// TIA Portal V17 export
// export: Created 2025-03-05T07:59:00.9677921Z, ExportSetting WithDefaults, DisplayName Totally Integrated Automation Portal, DisplayVersion V17 Update 8, DisplayName TIA Portal Openness, DisplayVersion V17 Update 8, DisplayName TIA Portal Version Control Interface, DisplayVersion V17, DisplayName SINAMICS Startdrive Advanced, DisplayVersion V17 SP2, DisplayName SINAMICS Startdrive G110M, G120, G120C, G120D, G120P, G115D, DisplayVersion V17 SP2, DisplayName SINAMICS Startdrive G130, G150, S120, S150, SINAMICS MV, S210, DisplayVersion V17 SP2, DisplayName STEP 7 Professional, DisplayVersion V17 Update 8, DisplayName SINUMERIK ONE STEP 7 Toolbox, DisplayVersion V17 Update 12, DisplayName SINUMERIK 840D sl STEP 7 Toolbox, DisplayVersion V17 Update 12, DisplayName STEP 7 Safety, DisplayVersion V17 Update 6, DisplayName WinCC Advanced, DisplayVersion V17 Update 8
DATA_BLOCK "DB2420_CNC_PLC_SIGNALS"   // DB2420
{ S7_Optimized_Access := 'FALSE'; DB_Accessible_From_OPC_UA := 'FALSE' }
AUTHOR : ETXETAR
VERSION : 1.0
// stored: AutoNumber false, DBAccessibleFromOPCUA false, DBAccessibleFromWebserver true, IsOnlyStoredInLoadMemory false, IsWriteProtectedInAS false
   VAR RETAIN
      NC_PLC_SIGNALS_1_32 : Struct   // NCK INPUTS EXTENSION BIT 41-72 / NC PLC SIGNALS BIT 1-32
         NC_PLC_SIGNAL_1 : Bool;   // NCK INPUTS EXTENSION 41 / UNIT 1 FIXTURE 1 GRIPPER CLOSED
         NC_PLC_SIGNAL_2 : Bool;   // NCK INPUTS EXTENSION 42 / UNIT 1 FIXTURE 1 GRIPPER OPEN
         NC_PLC_SIGNAL_3 : Bool;   // NCK INPUTS EXTENSION 43 / UNIT 1 FIXTURE 1 GRIPPER LOW
         NC_PLC_SIGNAL_4 : Bool;   // NCK INPUTS EXTENSION 44
         NC_PLC_SIGNAL_5 : Bool;   // NCK INPUTS EXTENSION 45
         NC_PLC_SIGNAL_6 : Bool;   // NCK INPUTS EXTENSION 46
         NC_PLC_SIGNAL_7 : Bool;   // NCK INPUTS EXTENSION 47
         NC_PLC_SIGNAL_8 : Bool;   // NCK INPUTS EXTENSION 48
         NC_PLC_SIGNAL_9 : Bool;   // NCK INPUTS EXTENSION 49
         NC_PLC_SIGNAL_10 : Bool;   // NCK INPUTS EXTENSION 50
         NC_PLC_SIGNAL_11 : Bool;   // NCK INPUTS EXTENSION 51
         NC_PLC_SIGNAL_12 : Bool;   // NCK INPUTS EXTENSION 52
         NC_PLC_SIGNAL_13 : Bool;   // NCK INPUTS EXTENSION 53
         NC_PLC_SIGNAL_14 : Bool;   // NCK INPUTS EXTENSION 54
         NC_PLC_SIGNAL_15 : Bool;   // NCK INPUTS EXTENSION 55
         NC_PLC_SIGNAL_16 : Bool;   // NCK INPUTS EXTENSION 56
         NC_PLC_SIGNAL_17 : Bool;   // NCK INPUTS EXTENSION 57 / UNIT 1 FIXTURE 2 GRIPPER CLOSED
         NC_PLC_SIGNAL_18 : Bool;   // NCK INPUTS EXTENSION 58 / UNIT 1 FIXTURE 2 GRIPPER OPEN
         NC_PLC_SIGNAL_19 : Bool;   // NCK INPUTS EXTENSION 59 / UNIT 1 FIXTURE 2 GRIPPER LOW
         NC_PLC_SIGNAL_20 : Bool;   // NCK INPUTS EXTENSION 60
         NC_PLC_SIGNAL_21 : Bool;   // NCK INPUTS EXTENSION 61
         NC_PLC_SIGNAL_22 : Bool;   // NCK INPUTS EXTENSION 62
         NC_PLC_SIGNAL_23 : Bool;   // NCK INPUTS EXTENSION 63
         NC_PLC_SIGNAL_24 : Bool;   // NCK INPUTS EXTENSION 64
         NC_PLC_SIGNAL_25 : Bool;   // NCK INPUTS EXTENSION 65
         NC_PLC_SIGNAL_26 : Bool;   // NCK INPUTS EXTENSION 66
         NC_PLC_SIGNAL_27 : Bool;   // NCK INPUTS EXTENSION 67
         NC_PLC_SIGNAL_28 : Bool;   // NCK INPUTS EXTENSION 68
         NC_PLC_SIGNAL_29 : Bool;   // NCK INPUTS EXTENSION 69
         NC_PLC_SIGNAL_30 : Bool;   // NCK INPUTS EXTENSION 70
         NC_PLC_SIGNAL_31 : Bool;   // NCK INPUTS EXTENSION 71
         NC_PLC_SIGNAL_32 : Bool;   // NCK INPUTS EXTENSION 72
      END_STRUCT;
      NC_PLC_SIGNALS_33_64 : Struct   // NCK INPUTS EXTENSION BIT 73-104 / NC PLC SIGNALS BIT 33-64
         NC_PLC_SIGNAL_33 : Bool;   // NCK INPUTS EXTENSION 73 / UNIT 1 FIXTURE 3 GRIPPER CLOSED
         NC_PLC_SIGNAL_34 : Bool;   // NCK INPUTS EXTENSION 74 / UNIT 1 FIXTURE 3 GRIPPER OPEN
         NC_PLC_SIGNAL_35 : Bool;   // NCK INPUTS EXTENSION 75 / UNIT 1 FIXTURE 3 GRIPPER LOW
         NC_PLC_SIGNAL_36 : Bool;   // NCK INPUTS EXTENSION 76
         NC_PLC_SIGNAL_37 : Bool;   // NCK INPUTS EXTENSION 77
         NC_PLC_SIGNAL_38 : Bool;   // NCK INPUTS EXTENSION 78
         NC_PLC_SIGNAL_39 : Bool;   // NCK INPUTS EXTENSION 79
         NC_PLC_SIGNAL_40 : Bool;   // NCK INPUTS EXTENSION 80
         NC_PLC_SIGNAL_41 : Bool;   // NCK INPUTS EXTENSION 81
         NC_PLC_SIGNAL_42 : Bool;   // NCK INPUTS EXTENSION 82
         NC_PLC_SIGNAL_43 : Bool;   // NCK INPUTS EXTENSION 83
         NC_PLC_SIGNAL_44 : Bool;   // NCK INPUTS EXTENSION 84
         NC_PLC_SIGNAL_45 : Bool;   // NCK INPUTS EXTENSION 85
         NC_PLC_SIGNAL_46 : Bool;   // NCK INPUTS EXTENSION 86
         NC_PLC_SIGNAL_47 : Bool;   // NCK INPUTS EXTENSION 87
         NC_PLC_SIGNAL_48 : Bool;   // NCK INPUTS EXTENSION 88
         NC_PLC_SIGNAL_49 : Bool;   // NCK INPUTS EXTENSION 89 / UNIT 1 FIXTURE 4 GRIPPER CLOSED
         NC_PLC_SIGNAL_50 : Bool;   // NCK INPUTS EXTENSION 90 / UNIT 1 FIXTURE 4 GRIPPER OPEN
         NC_PLC_SIGNAL_51 : Bool;   // NCK INPUTS EXTENSION 91 / UNIT 1 FIXTURE 4 GRIPPER LOW
         NC_PLC_SIGNAL_52 : Bool;   // NCK INPUTS EXTENSION 92
         NC_PLC_SIGNAL_53 : Bool;   // NCK INPUTS EXTENSION 93
         NC_PLC_SIGNAL_54 : Bool;   // NCK INPUTS EXTENSION 94
         NC_PLC_SIGNAL_55 : Bool;   // NCK INPUTS EXTENSION 95
         NC_PLC_SIGNAL_56 : Bool;   // NCK INPUTS EXTENSION 96
         NC_PLC_SIGNAL_57 : Bool;   // NCK INPUTS EXTENSION 97
         NC_PLC_SIGNAL_58 : Bool;   // NCK INPUTS EXTENSION 98
         NC_PLC_SIGNAL_59 : Bool;   // NCK INPUTS EXTENSION 99
         NC_PLC_SIGNAL_60 : Bool;   // NCK INPUTS EXTENSION 100
         NC_PLC_SIGNAL_61 : Bool;   // NCK INPUTS EXTENSION 101
         NC_PLC_SIGNAL_62 : Bool;   // NCK INPUTS EXTENSION 102
         NC_PLC_SIGNAL_63 : Bool;   // NCK INPUTS EXTENSION 103
         NC_PLC_SIGNAL_64 : Bool;   // NCK INPUTS EXTENSION 104
      END_STRUCT;
      NC_PLC_SIGNALS_65_96 : Struct   // NCK INPUTS EXTENSION BIT 73-104 / NC PLC SIGNALS BIT 65-96
         NC_PLC_SIGNAL_65 : Bool;   // NCK INPUTS EXTENSION 73 / UNIT 2 FIXTURE 1 GRIPPER CLOSED
         NC_PLC_SIGNAL_66 : Bool;   // NCK INPUTS EXTENSION 74 / UNIT 2 FIXTURE 1 GRIPPER OPEN
         NC_PLC_SIGNAL_67 : Bool;   // NCK INPUTS EXTENSION 75 / UNIT 2 FIXTURE 1 GRIPPER LOW
         NC_PLC_SIGNAL_68 : Bool;   // NCK INPUTS EXTENSION 76
         NC_PLC_SIGNAL_69 : Bool;   // NCK INPUTS EXTENSION 77
         NC_PLC_SIGNAL_70 : Bool;   // NCK INPUTS EXTENSION 78
         NC_PLC_SIGNAL_71 : Bool;   // NCK INPUTS EXTENSION 79
         NC_PLC_SIGNAL_72 : Bool;   // NCK INPUTS EXTENSION 80
         NC_PLC_SIGNAL_73 : Bool;   // NCK INPUTS EXTENSION 81
         NC_PLC_SIGNAL_74 : Bool;   // NCK INPUTS EXTENSION 82
         NC_PLC_SIGNAL_75 : Bool;   // NCK INPUTS EXTENSION 83
         NC_PLC_SIGNAL_76 : Bool;   // NCK INPUTS EXTENSION 84
         NC_PLC_SIGNAL_77 : Bool;   // NCK INPUTS EXTENSION 85
         NC_PLC_SIGNAL_78 : Bool;   // NCK INPUTS EXTENSION 86
         NC_PLC_SIGNAL_79 : Bool;   // NCK INPUTS EXTENSION 87
         NC_PLC_SIGNAL_80 : Bool;   // NCK INPUTS EXTENSION 88
         NC_PLC_SIGNAL_81 : Bool;   // NCK INPUTS EXTENSION 89 / UNIT 2 FIXTURE 2 GRIPPER CLOSED
         NC_PLC_SIGNAL_82 : Bool;   // NCK INPUTS EXTENSION 90 / UNIT 2 FIXTURE 2 GRIPPER OPEN
         NC_PLC_SIGNAL_83 : Bool;   // NCK INPUTS EXTENSION 91 / UNIT 2 FIXTURE 2 GRIPPER LOW
         NC_PLC_SIGNAL_84 : Bool;   // NCK INPUTS EXTENSION 92
         NC_PLC_SIGNAL_85 : Bool;   // NCK INPUTS EXTENSION 93
         NC_PLC_SIGNAL_86 : Bool;   // NCK INPUTS EXTENSION 94
         NC_PLC_SIGNAL_87 : Bool;   // NCK INPUTS EXTENSION 95
         NC_PLC_SIGNAL_88 : Bool;   // NCK INPUTS EXTENSION 96
         NC_PLC_SIGNAL_89 : Bool;   // NCK INPUTS EXTENSION 97
         NC_PLC_SIGNAL_90 : Bool;   // NCK INPUTS EXTENSION 98
         NC_PLC_SIGNAL_91 : Bool;   // NCK INPUTS EXTENSION 99
         NC_PLC_SIGNAL_92 : Bool;   // NCK INPUTS EXTENSION 100
         NC_PLC_SIGNAL_93 : Bool;   // NCK INPUTS EXTENSION 101
         NC_PLC_SIGNAL_94 : Bool;   // NCK INPUTS EXTENSION 102
         NC_PLC_SIGNAL_95 : Bool;   // NCK INPUTS EXTENSION 103
         NC_PLC_SIGNAL_96 : Bool;   // NCK INPUTS EXTENSION 104
      END_STRUCT;
      NC_PLC_SIGNALS_97_128 : Struct   // NCK INPUTS EXTENSION BIT 73-104 / NC PLC SIGNALS BIT 97-128
         NC_PLC_SIGNAL_97 : Bool;   // NCK INPUTS EXTENSION 73 / UNIT 2 FIXTURE 3 GRIPPER CLOSED
         NC_PLC_SIGNAL_98 : Bool;   // NCK INPUTS EXTENSION 74 / UNIT 2 FIXTURE 3 GRIPPER OPEN
         NC_PLC_SIGNAL_99 : Bool;   // NCK INPUTS EXTENSION 75 / UNIT 2 FIXTURE 3 GRIPPER LOW
         NC_PLC_SIGNAL_100 : Bool;   // NCK INPUTS EXTENSION 76
         NC_PLC_SIGNAL_101 : Bool;   // NCK INPUTS EXTENSION 77
         NC_PLC_SIGNAL_102 : Bool;   // NCK INPUTS EXTENSION 78
         NC_PLC_SIGNAL_103 : Bool;   // NCK INPUTS EXTENSION 79
         NC_PLC_SIGNAL_104 : Bool;   // NCK INPUTS EXTENSION 80
         NC_PLC_SIGNAL_105 : Bool;   // NCK INPUTS EXTENSION 81
         NC_PLC_SIGNAL_106 : Bool;   // NCK INPUTS EXTENSION 82
         NC_PLC_SIGNAL_107 : Bool;   // NCK INPUTS EXTENSION 83
         NC_PLC_SIGNAL_108 : Bool;   // NCK INPUTS EXTENSION 84
         NC_PLC_SIGNAL_109 : Bool;   // NCK INPUTS EXTENSION 85
         NC_PLC_SIGNAL_110 : Bool;   // NCK INPUTS EXTENSION 86
         NC_PLC_SIGNAL_111 : Bool;   // NCK INPUTS EXTENSION 87
         NC_PLC_SIGNAL_112 : Bool;   // NCK INPUTS EXTENSION 88
         NC_PLC_SIGNAL_113 : Bool;   // NCK INPUTS EXTENSION 89 / UNIT 2 FIXTURE 4 GRIPPER CLOSED
         NC_PLC_SIGNAL_114 : Bool;   // NCK INPUTS EXTENSION 90 / UNIT 2 FIXTURE 4 GRIPPER OPEN
         NC_PLC_SIGNAL_115 : Bool;   // NCK INPUTS EXTENSION 91 / UNIT 2 FIXTURE 4 GRIPPER LOW
         NC_PLC_SIGNAL_116 : Bool;   // NCK INPUTS EXTENSION 92
         NC_PLC_SIGNAL_117 : Bool;   // NCK INPUTS EXTENSION 93
         NC_PLC_SIGNAL_118 : Bool;   // NCK INPUTS EXTENSION 94
         NC_PLC_SIGNAL_119 : Bool;   // NCK INPUTS EXTENSION 95
         NC_PLC_SIGNAL_120 : Bool;   // NCK INPUTS EXTENSION 96
         NC_PLC_SIGNAL_121 : Bool;   // NCK INPUTS EXTENSION 97
         NC_PLC_SIGNAL_122 : Bool;   // NCK INPUTS EXTENSION 98
         NC_PLC_SIGNAL_123 : Bool;   // NCK INPUTS EXTENSION 99
         NC_PLC_SIGNAL_124 : Bool;   // NCK INPUTS EXTENSION 100
         NC_PLC_SIGNAL_125 : Bool;   // NCK INPUTS EXTENSION 101
         NC_PLC_SIGNAL_126 : Bool;   // NCK INPUTS EXTENSION 102
         NC_PLC_SIGNAL_127 : Bool;   // NCK INPUTS EXTENSION 103
         NC_PLC_SIGNAL_128 : Bool;   // NCK INPUTS EXTENSION 104
      END_STRUCT;
      NC_PLC_SIGNALS_129_160 : Struct   // NCK INPUTS EXTENSION BIT 73-104 / NC PLC SIGNALS BIT 129-160
         NC_PLC_SIGNAL_129 : Bool;   // NCK INPUTS EXTENSION 73 / NC PLC SIGNAL 129
         NC_PLC_SIGNAL_130 : Bool;   // NCK INPUTS EXTENSION 74 / NC PLC SIGNAL 130
         NC_PLC_SIGNAL_131 : Bool;   // NCK INPUTS EXTENSION 75 / NC PLC SIGNAL 131
         NC_PLC_SIGNAL_132 : Bool;   // NCK INPUTS EXTENSION 76 / NC PLC SIGNAL 132
         NC_PLC_SIGNAL_133 : Bool;   // NCK INPUTS EXTENSION 77 / NC PLC SIGNAL 133
         NC_PLC_SIGNAL_134 : Bool;   // NCK INPUTS EXTENSION 78 / NC PLC SIGNAL 134
         NC_PLC_SIGNAL_135 : Bool;   // NCK INPUTS EXTENSION 79 / NC PLC SIGNAL 135
         NC_PLC_SIGNAL_136 : Bool;   // NCK INPUTS EXTENSION 80 / NC PLC SIGNAL 136
         NC_PLC_SIGNAL_137 : Bool;   // NCK INPUTS EXTENSION 81 / NC PLC SIGNAL 137
         NC_PLC_SIGNAL_138 : Bool;   // NCK INPUTS EXTENSION 82 / NC PLC SIGNAL 138
         NC_PLC_SIGNAL_139 : Bool;   // NCK INPUTS EXTENSION 83 / NC PLC SIGNAL 139
         NC_PLC_SIGNAL_140 : Bool;   // NCK INPUTS EXTENSION 84 / NC PLC SIGNAL 140
         NC_PLC_SIGNAL_141 : Bool;   // NCK INPUTS EXTENSION 85 / NC PLC SIGNAL 141
         NC_PLC_SIGNAL_142 : Bool;   // NCK INPUTS EXTENSION 86 / NC PLC SIGNAL 142
         NC_PLC_SIGNAL_143 : Bool;   // NCK INPUTS EXTENSION 87 / NC PLC SIGNAL 143
         NC_PLC_SIGNAL_144 : Bool;   // NCK INPUTS EXTENSION 88 / NC PLC SIGNAL 144
         NC_PLC_SIGNAL_145 : Bool;   // NCK INPUTS EXTENSION 89 / NC PLC SIGNAL 145
         NC_PLC_SIGNAL_146 : Bool;   // NCK INPUTS EXTENSION 90 / NC PLC SIGNAL 146
         NC_PLC_SIGNAL_147 : Bool;   // NCK INPUTS EXTENSION 91 / NC PLC SIGNAL 147
         NC_PLC_SIGNAL_148 : Bool;   // NCK INPUTS EXTENSION 92 / NC PLC SIGNAL 148
         NC_PLC_SIGNAL_149 : Bool;   // NCK INPUTS EXTENSION 93 / NC PLC SIGNAL 149
         NC_PLC_SIGNAL_150 : Bool;   // NCK INPUTS EXTENSION 94 / NC PLC SIGNAL 150
         NC_PLC_SIGNAL_151 : Bool;   // NCK INPUTS EXTENSION 95 / NC PLC SIGNAL 151
         NC_PLC_SIGNAL_152 : Bool;   // NCK INPUTS EXTENSION 96 / NC PLC SIGNAL 152
         NC_PLC_SIGNAL_153 : Bool;   // NCK INPUTS EXTENSION 97 / NC PLC SIGNAL 153
         NC_PLC_SIGNAL_154 : Bool;   // NCK INPUTS EXTENSION 98 / NC PLC SIGNAL 154
         NC_PLC_SIGNAL_155 : Bool;   // NCK INPUTS EXTENSION 99 / NC PLC SIGNAL 155
         NC_PLC_SIGNAL_156 : Bool;   // NCK INPUTS EXTENSION 100 / NC PLC SIGNAL 156
         NC_PLC_SIGNAL_157 : Bool;   // NCK INPUTS EXTENSION 101 / NC PLC SIGNAL 157
         NC_PLC_SIGNAL_158 : Bool;   // NCK INPUTS EXTENSION 102 / NC PLC SIGNAL 158
         NC_PLC_SIGNAL_159 : Bool;   // NCK INPUTS EXTENSION 103 / NC PLC SIGNAL 159
         NC_PLC_SIGNAL_160 : Bool;   // NCK INPUTS EXTENSION 104 / NC PLC SIGNAL 160
      END_STRUCT;
      NC_PLC_SIGNALS_161_192 : Struct   // NCK INPUTS EXTENSION BIT 73-104 / NC PLC SIGNALS BIT 161-192
         NC_PLC_SIGNAL_161 : Bool;   // NCK INPUTS EXTENSION 73 / NC PLC SIGNAL 161
         NC_PLC_SIGNAL_162 : Bool;   // NCK INPUTS EXTENSION 74 / NC PLC SIGNAL 162
         NC_PLC_SIGNAL_163 : Bool;   // NCK INPUTS EXTENSION 75 / NC PLC SIGNAL 163
         NC_PLC_SIGNAL_164 : Bool;   // NCK INPUTS EXTENSION 76 / NC PLC SIGNAL 164
         NC_PLC_SIGNAL_165 : Bool;   // NCK INPUTS EXTENSION 77 / NC PLC SIGNAL 165
         NC_PLC_SIGNAL_166 : Bool;   // NCK INPUTS EXTENSION 78 / NC PLC SIGNAL 166
         NC_PLC_SIGNAL_167 : Bool;   // NCK INPUTS EXTENSION 79 / NC PLC SIGNAL 167
         NC_PLC_SIGNAL_168 : Bool;   // NCK INPUTS EXTENSION 80 / NC PLC SIGNAL 168
         NC_PLC_SIGNAL_169 : Bool;   // NCK INPUTS EXTENSION 81 / NC PLC SIGNAL 169
         NC_PLC_SIGNAL_170 : Bool;   // NCK INPUTS EXTENSION 82 / NC PLC SIGNAL 170
         NC_PLC_SIGNAL_171 : Bool;   // NCK INPUTS EXTENSION 83 / NC PLC SIGNAL 171
         NC_PLC_SIGNAL_172 : Bool;   // NCK INPUTS EXTENSION 84 / NC PLC SIGNAL 172
         NC_PLC_SIGNAL_173 : Bool;   // NCK INPUTS EXTENSION 85 / NC PLC SIGNAL 173
         NC_PLC_SIGNAL_174 : Bool;   // NCK INPUTS EXTENSION 86 / NC PLC SIGNAL 174
         NC_PLC_SIGNAL_175 : Bool;   // NCK INPUTS EXTENSION 87 / NC PLC SIGNAL 175
         NC_PLC_SIGNAL_176 : Bool;   // NCK INPUTS EXTENSION 88 / NC PLC SIGNAL 176
         NC_PLC_SIGNAL_177 : Bool;   // NCK INPUTS EXTENSION 89 / NC PLC SIGNAL 177
         NC_PLC_SIGNAL_178 : Bool;   // NCK INPUTS EXTENSION 90 / NC PLC SIGNAL 178
         NC_PLC_SIGNAL_179 : Bool;   // NCK INPUTS EXTENSION 91 / NC PLC SIGNAL 179
         NC_PLC_SIGNAL_180 : Bool;   // NCK INPUTS EXTENSION 92 / NC PLC SIGNAL 180
         NC_PLC_SIGNAL_181 : Bool;   // NCK INPUTS EXTENSION 93 / NC PLC SIGNAL 181
         NC_PLC_SIGNAL_182 : Bool;   // NCK INPUTS EXTENSION 94 / NC PLC SIGNAL 182
         NC_PLC_SIGNAL_183 : Bool;   // NCK INPUTS EXTENSION 95 / NC PLC SIGNAL 183
         NC_PLC_SIGNAL_184 : Bool;   // NCK INPUTS EXTENSION 96 / NC PLC SIGNAL 184
         NC_PLC_SIGNAL_185 : Bool;   // NCK INPUTS EXTENSION 97 / NC PLC SIGNAL 185
         NC_PLC_SIGNAL_186 : Bool;   // NCK INPUTS EXTENSION 98 / NC PLC SIGNAL 186
         NC_PLC_SIGNAL_187 : Bool;   // NCK INPUTS EXTENSION 99 / NC PLC SIGNAL 187
         NC_PLC_SIGNAL_188 : Bool;   // NCK INPUTS EXTENSION 100 / NC PLC SIGNAL 188
         NC_PLC_SIGNAL_189 : Bool;   // NCK INPUTS EXTENSION 101 / NC PLC SIGNAL 189
         NC_PLC_SIGNAL_190 : Bool;   // NCK INPUTS EXTENSION 102 / NC PLC SIGNAL 190
         NC_PLC_SIGNAL_191 : Bool;   // NCK INPUTS EXTENSION 103 / NC PLC SIGNAL 191
         NC_PLC_SIGNAL_192 : Bool;   // NCK INPUTS EXTENSION 104 / NC PLC SIGNAL 192
      END_STRUCT;
      NC_PLC_SIGNALS_193_224 : Struct   // NCK INPUTS EXTENSION BIT 73-104 / NC PLC SIGNALS BIT 193-224
         NC_PLC_SIGNAL_193 : Bool;   // NCK INPUTS EXTENSION 73 / NC PLC SIGNAL 193
         NC_PLC_SIGNAL_194 : Bool;   // NCK INPUTS EXTENSION 74 / NC PLC SIGNAL 194
         NC_PLC_SIGNAL_195 : Bool;   // NCK INPUTS EXTENSION 75 / NC PLC SIGNAL 195
         NC_PLC_SIGNAL_196 : Bool;   // NCK INPUTS EXTENSION 76 / NC PLC SIGNAL 196
         NC_PLC_SIGNAL_197 : Bool;   // NCK INPUTS EXTENSION 77 / NC PLC SIGNAL 197
         NC_PLC_SIGNAL_198 : Bool;   // NCK INPUTS EXTENSION 78 / NC PLC SIGNAL 198
         NC_PLC_SIGNAL_199 : Bool;   // NCK INPUTS EXTENSION 79 / NC PLC SIGNAL 199
         NC_PLC_SIGNAL_200 : Bool;   // NCK INPUTS EXTENSION 80 / NC PLC SIGNAL 200
         NC_PLC_SIGNAL_201 : Bool;   // NCK INPUTS EXTENSION 81 / NC PLC SIGNAL 201
         NC_PLC_SIGNAL_202 : Bool;   // NCK INPUTS EXTENSION 82 / NC PLC SIGNAL 202
         NC_PLC_SIGNAL_203 : Bool;   // NCK INPUTS EXTENSION 83 / NC PLC SIGNAL 203
         NC_PLC_SIGNAL_204 : Bool;   // NCK INPUTS EXTENSION 84 / NC PLC SIGNAL 204
         NC_PLC_SIGNAL_205 : Bool;   // NCK INPUTS EXTENSION 85 / NC PLC SIGNAL 205
         NC_PLC_SIGNAL_206 : Bool;   // NCK INPUTS EXTENSION 86 / NC PLC SIGNAL 206
         NC_PLC_SIGNAL_207 : Bool;   // NCK INPUTS EXTENSION 87 / NC PLC SIGNAL 207
         NC_PLC_SIGNAL_208 : Bool;   // NCK INPUTS EXTENSION 88 / NC PLC SIGNAL 208
         NC_PLC_SIGNAL_209 : Bool;   // NCK INPUTS EXTENSION 89 / NC PLC SIGNAL 209
         NC_PLC_SIGNAL_210 : Bool;   // NCK INPUTS EXTENSION 90 / NC PLC SIGNAL 210
         NC_PLC_SIGNAL_211 : Bool;   // NCK INPUTS EXTENSION 91 / NC PLC SIGNAL 211
         NC_PLC_SIGNAL_212 : Bool;   // NCK INPUTS EXTENSION 92 / NC PLC SIGNAL 212
         NC_PLC_SIGNAL_213 : Bool;   // NCK INPUTS EXTENSION 93 / NC PLC SIGNAL 213
         NC_PLC_SIGNAL_214 : Bool;   // NCK INPUTS EXTENSION 94 / NC PLC SIGNAL 214
         NC_PLC_SIGNAL_215 : Bool;   // NCK INPUTS EXTENSION 95 / NC PLC SIGNAL 215
         NC_PLC_SIGNAL_216 : Bool;   // NCK INPUTS EXTENSION 96 / NC PLC SIGNAL 216
         NC_PLC_SIGNAL_217 : Bool;   // NCK INPUTS EXTENSION 97 / NC PLC SIGNAL 217
         NC_PLC_SIGNAL_218 : Bool;   // NCK INPUTS EXTENSION 98 / NC PLC SIGNAL 218
         NC_PLC_SIGNAL_219 : Bool;   // NCK INPUTS EXTENSION 99 / NC PLC SIGNAL 219
         NC_PLC_SIGNAL_220 : Bool;   // NCK INPUTS EXTENSION 100 / NC PLC SIGNAL 220
         NC_PLC_SIGNAL_221 : Bool;   // NCK INPUTS EXTENSION 101 / NC PLC SIGNAL 221
         NC_PLC_SIGNAL_222 : Bool;   // NCK INPUTS EXTENSION 102 / NC PLC SIGNAL 222
         NC_PLC_SIGNAL_223 : Bool;   // NCK INPUTS EXTENSION 103 / NC PLC SIGNAL 223
         NC_PLC_SIGNAL_224 : Bool;   // NCK INPUTS EXTENSION 104 / NC PLC SIGNAL 224
      END_STRUCT;
      NC_PLC_SIGNALS_225_256 : Struct   // NCK INPUTS EXTENSION BIT 73-104 / NC PLC SIGNALS BIT 225-256
         NC_PLC_SIGNAL_225 : Bool;   // NCK INPUTS EXTENSION 73 / NC PLC SIGNAL 225
         NC_PLC_SIGNAL_226 : Bool;   // NCK INPUTS EXTENSION 74 / NC PLC SIGNAL 226
         NC_PLC_SIGNAL_227 : Bool;   // NCK INPUTS EXTENSION 75 / NC PLC SIGNAL 227
         NC_PLC_SIGNAL_228 : Bool;   // NCK INPUTS EXTENSION 76 / NC PLC SIGNAL 228
         NC_PLC_SIGNAL_229 : Bool;   // NCK INPUTS EXTENSION 77 / NC PLC SIGNAL 229
         NC_PLC_SIGNAL_230 : Bool;   // NCK INPUTS EXTENSION 78 / NC PLC SIGNAL 230
         NC_PLC_SIGNAL_231 : Bool;   // NCK INPUTS EXTENSION 79 / NC PLC SIGNAL 231
         NC_PLC_SIGNAL_232 : Bool;   // NCK INPUTS EXTENSION 80 / NC PLC SIGNAL 232
         NC_PLC_SIGNAL_233 : Bool;   // NCK INPUTS EXTENSION 81 / NC PLC SIGNAL 233
         NC_PLC_SIGNAL_234 : Bool;   // NCK INPUTS EXTENSION 82 / NC PLC SIGNAL 234
         NC_PLC_SIGNAL_235 : Bool;   // NCK INPUTS EXTENSION 83 / NC PLC SIGNAL 235
         NC_PLC_SIGNAL_236 : Bool;   // NCK INPUTS EXTENSION 84 / NC PLC SIGNAL 236
         NC_PLC_SIGNAL_237 : Bool;   // NCK INPUTS EXTENSION 85 / NC PLC SIGNAL 237
         NC_PLC_SIGNAL_238 : Bool;   // NCK INPUTS EXTENSION 86 / NC PLC SIGNAL 238
         NC_PLC_SIGNAL_239 : Bool;   // NCK INPUTS EXTENSION 87 / NC PLC SIGNAL 239
         NC_PLC_SIGNAL_240 : Bool;   // NCK INPUTS EXTENSION 88 / NC PLC SIGNAL 240
         NC_PLC_SIGNAL_241 : Bool;   // NCK INPUTS EXTENSION 89 / NC PLC SIGNAL 241
         NC_PLC_SIGNAL_242 : Bool;   // NCK INPUTS EXTENSION 90 / NC PLC SIGNAL 242
         NC_PLC_SIGNAL_243 : Bool;   // NCK INPUTS EXTENSION 91 / NC PLC SIGNAL 243
         NC_PLC_SIGNAL_244 : Bool;   // NCK INPUTS EXTENSION 92 / NC PLC SIGNAL 244
         NC_PLC_SIGNAL_245 : Bool;   // NCK INPUTS EXTENSION 93 / NC PLC SIGNAL 245
         NC_PLC_SIGNAL_246 : Bool;   // NCK INPUTS EXTENSION 94 / NC PLC SIGNAL 246
         NC_PLC_SIGNAL_247 : Bool;   // NCK INPUTS EXTENSION 95 / NC PLC SIGNAL 247
         NC_PLC_SIGNAL_248 : Bool;   // NCK INPUTS EXTENSION 96 / NC PLC SIGNAL 248
         NC_PLC_SIGNAL_249 : Bool;   // NCK INPUTS EXTENSION 97 / NC PLC SIGNAL 249
         NC_PLC_SIGNAL_250 : Bool;   // NCK INPUTS EXTENSION 98 / NC PLC SIGNAL 250
         NC_PLC_SIGNAL_251 : Bool;   // NCK INPUTS EXTENSION 99 / NC PLC SIGNAL 251
         NC_PLC_SIGNAL_252 : Bool;   // NCK INPUTS EXTENSION 100 / NC PLC SIGNAL 252
         NC_PLC_SIGNAL_253 : Bool;   // NCK INPUTS EXTENSION 101 / NC PLC SIGNAL 253
         NC_PLC_SIGNAL_254 : Bool;   // NCK INPUTS EXTENSION 102 / NC PLC SIGNAL 254
         NC_PLC_SIGNAL_255 : Bool;   // NCK INPUTS EXTENSION 103 / NC PLC SIGNAL 255
         NC_PLC_SIGNAL_256 : Bool;   // NCK INPUTS EXTENSION 104 / NC PLC SIGNAL 256
      END_STRUCT;
      DBB_DBW_DBD_VAL_4040 : Int := 4040;   // NCK INPUTS EXTENSION BIT 41-72 / NC PLC SIGNALS BIT 1-32
      DBB_DBW_DBD_VAL_4041 : Int := 4041;
      DBB_DBW_DBD_VAL_4042 : Int := 4042;
      DBB_DBW_DBD_VAL_4043 : Int := 4043;
      DBB_DBW_DBD_VAL_4044 : Int := 4044;   // NCK INPUTS EXTENSION BIT 73-104 / NC PLC SIGNALS BIT 33-64
      DBB_DBW_DBD_VAL_4045 : Int := 4045;
      DBB_DBW_DBD_VAL_4046 : Int := 4046;
      DBB_DBW_DBD_VAL_4047 : Int := 4047;
      DBB_DBW_DBD_VAL_4048 : Int := 4048;   // NC PLC SIGNALS BIT 65-96
      DBB_DBW_DBD_VAL_4049 : Int := 4049;
      DBB_DBW_DBD_VAL_4050 : Int := 4050;
      DBB_DBW_DBD_VAL_4051 : Int := 4051;
      DBB_DBW_DBD_VAL_4052 : Int := 4052;   // NC PLC SIGNALS BIT 97-128
      DBB_DBW_DBD_VAL_4053 : Int := 4053;
      DBB_DBW_DBD_VAL_4054 : Int := 4054;
      DBB_DBW_DBD_VAL_4055 : Int := 4055;
      DBB_DBW_DBD_VAL_4056 : Int := 4056;   // NC PLC SIGNALS BIT 129-160
      DBB_DBW_DBD_VAL_4057 : Int := 4057;
      DBB_DBW_DBD_VAL_4058 : Int := 4058;
      DBB_DBW_DBD_VAL_4059 : Int := 4059;
      DBB_DBW_DBD_VAL_4060 : Int := 4060;   // NC PLC SIGNALS BIT 161-192
      DBB_DBW_DBD_VAL_4061 : Int := 4061;
      DBB_DBW_DBD_VAL_4062 : Int := 4062;
      DBB_DBW_DBD_VAL_4063 : Int := 4063;
      DBB_DBW_DBD_VAL_4064 : Int := 4064;   // NC PLC SIGNALS BIT 193-224
      DBB_DBW_DBD_VAL_4065 : Int := 4065;
      DBB_DBW_DBD_VAL_4066 : Int := 4066;
      DBB_DBW_DBD_VAL_4067 : Int := 4067;
      DBB_DBW_DBD_VAL_4068 : Int := 4068;   // NC PLC SIGNALS BIT 225-256
      DBB_DBW_DBD_VAL_4069 : Int := 4069;
      DBB_DBW_DBD_VAL_4070 : Int := 4070;
      DBB_DBW_DBD_VAL_4071 : Int := 4071;
   END_VAR
BEGIN
END_DATA_BLOCK
